ADAPTER Adapter_Handshake (* Adapter Interface *)
  (* Standard: 61499-1 *)
  (* Version 0.0, 11/2/2020, prana, nxtControl GmbH *)
  PACKAGE Main;
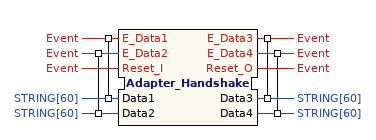
  EVENT_INPUT
    E_Data1 WITH Data1;
    E_Data2 WITH Data2;
    Reset_I;
  END_EVENT
  EVENT_OUTPUT
    E_Data3 WITH Data3;
    E_Data4 WITH Data4;
    Reset_O;
  END_EVENT
  VAR_INPUT
    Data1 : STRING[60];
    Data2 : STRING[60];
  END_VAR
  VAR_OUTPUT
    Data3 : STRING[60];
    Data4 : STRING[60];
  END_VAR
  SERVICE SOCKET/PLUG
    SEQUENCE request_confirm
      SOCKET.REQ(REQD) -> PLUG.REQ(REQD);
      PLUG.CNF(CNFD) -> SOCKET.CNF(CNFD);
    END_SEQUENCE
    SEQUENCE indication_response
      PLUG.IND(INDD) -> SOCKET.IND(INDD);
      SOCKET.RSP(RSPD) -> PLUG.RSP(RSPD);
    END_SEQUENCE
  END_SERVICE
END_ADAPTER
